% RSLogix 500 project filling_station.RSS, saved by version 8.30.00.16 %
PROJECT "UNTITLED"    % processor: Bul.1763 MicroLogix 1100 Series B %

PROGRAM FILES
  LAD 2   4 rungs
  LAD 3 "IO"  8 rungs
  LAD 4 "STATE"  7 rungs
  LAD 5 "CONTROLS"  4 rungs

DATA FILES
  O0 OUTPUT  4 elements
  I1 INPUT  6 elements
  S2 STATUS  66 elements
  B3 BINARY  3 elements
  T4 TIMER  1 elements
  C5 COUNTER  1 elements
  R6 CONTROL  1 elements
  N7 INTEGER  10 elements
  F8 FLOAT  1 elements

LADDER 2
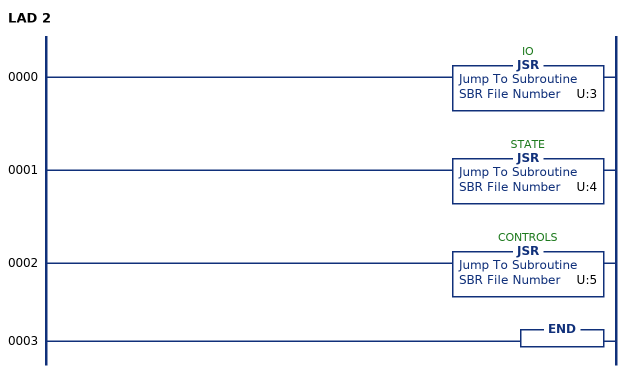
% Rung: 0 %
SOR JSR U:3 EOR
%   U:3  "IO" %
% Rung: 1 %
SOR JSR U:4 EOR
%   U:4  "STATE" %
% Rung: 2 %
SOR JSR U:5 EOR
%   U:5  "CONTROLS" %
% Rung: 3 %
SOR END EOR

LADDER 3 "IO"
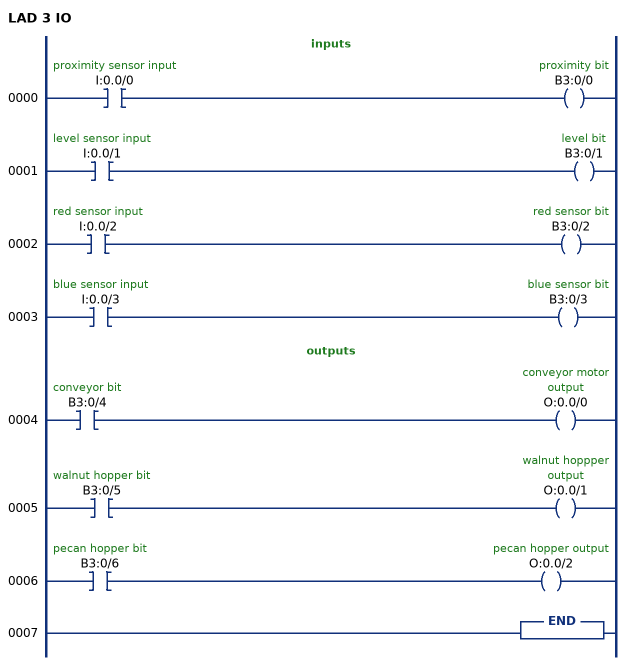
% Rung: 0 %
% TITLE: inputs %
SOR XIC I:0.0/0 OTE B3:0/0 EOR
%   I:0.0/0  "proximity sensor input" %
%   B3:0/0  "proximity bit" %
% Rung: 1 %
SOR XIC I:0.0/1 OTE B3:0/1 EOR
%   I:0.0/1  "level sensor input" %
%   B3:0/1  "level bit" %
% Rung: 2 %
SOR XIC I:0.0/2 OTE B3:0/2 EOR
%   I:0.0/2  "red sensor input" %
%   B3:0/2  "red sensor bit" %
% Rung: 3 %
SOR XIC I:0.0/3 OTE B3:0/3 EOR
%   I:0.0/3  "blue sensor input" %
%   B3:0/3  "blue sensor bit" %
% Rung: 4 %
% TITLE: outputs %
SOR XIC B3:0/4 OTE O:0.0/0 EOR
%   B3:0/4  "conveyor bit" %
%   O:0.0/0  "conveyor motor output" %
% Rung: 5 %
SOR XIC B3:0/5 OTE O:0.0/1 EOR
%   B3:0/5  "walnut hopper bit" %
%   O:0.0/1  "walnut hoppper output" %
% Rung: 6 %
SOR XIC B3:0/6 OTE O:0.0/2 EOR
%   B3:0/6  "pecan hopper bit" %
%   O:0.0/2  "pecan hopper output" %
% Rung: 7 %
SOR END EOR

LADDER 4 "STATE"
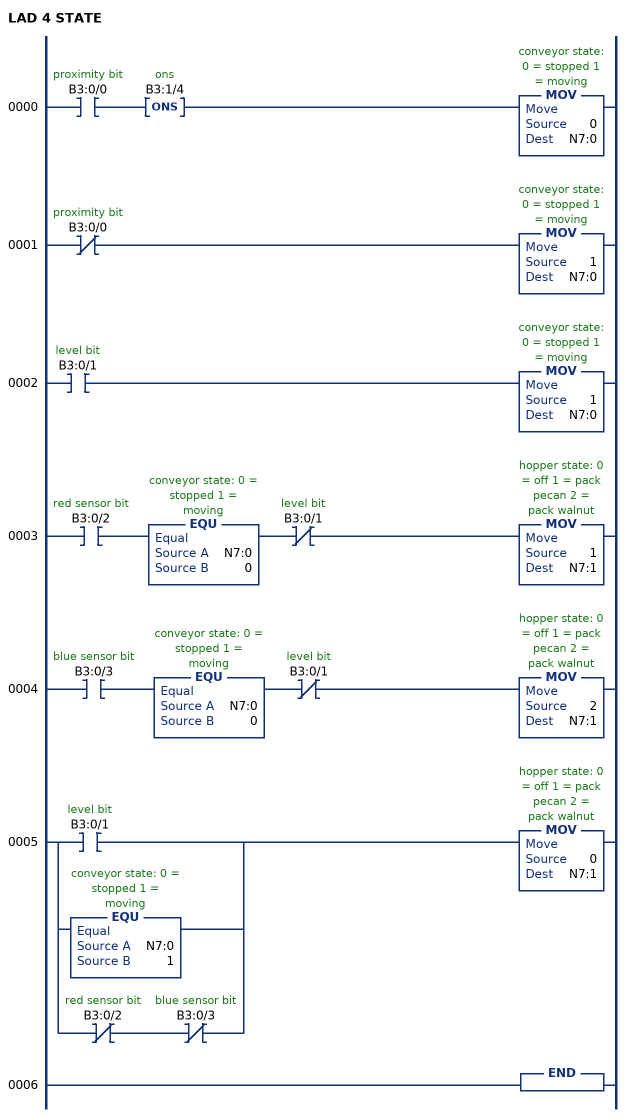
% Rung: 0 %
SOR XIC B3:0/0 ONS B3:1/4 MOV 0 N7:0 EOR
%   B3:0/0  "proximity bit" %
%   B3:1/4  "ons" %
%   N7:0  "conveyor state: 0 = stopped 1 = moving" %
% Rung: 1 %
SOR XIO B3:0/0 MOV 1 N7:0 EOR
%   B3:0/0  "proximity bit" %
%   N7:0  "conveyor state: 0 = stopped 1 = moving" %
% Rung: 2 %
SOR XIC B3:0/1 MOV 1 N7:0 EOR
%   B3:0/1  "level bit" %
%   N7:0  "conveyor state: 0 = stopped 1 = moving" %
% Rung: 3 %
SOR XIC B3:0/2 EQU N7:0 0 XIO B3:0/1 MOV 1 N7:1 EOR
%   B3:0/2  "red sensor bit" %
%   N7:0  "conveyor state: 0 = stopped 1 = moving" %
%   B3:0/1  "level bit" %
%   N7:1  "hopper state: 0 = off 1 = pack pecan 2 = pack walnut" %
% Rung: 4 %
SOR XIC B3:0/3 EQU N7:0 0 XIO B3:0/1 MOV 2 N7:1 EOR
%   B3:0/3  "blue sensor bit" %
%   N7:0  "conveyor state: 0 = stopped 1 = moving" %
%   B3:0/1  "level bit" %
%   N7:1  "hopper state: 0 = off 1 = pack pecan 2 = pack walnut" %
% Rung: 5 %  % edit flag set %
SOR BST XIC B3:0/1 NXB EQU N7:0 1 NXB XIO B3:0/2 XIO B3:0/3 BND MOV 0 N7:1 EOR
%   B3:0/1  "level bit" %
%   N7:0  "conveyor state: 0 = stopped 1 = moving" %
%   B3:0/2  "red sensor bit" %
%   B3:0/3  "blue sensor bit" %
%   N7:1  "hopper state: 0 = off 1 = pack pecan 2 = pack walnut" %
% Rung: 6 %
SOR END EOR

LADDER 5 "CONTROLS"
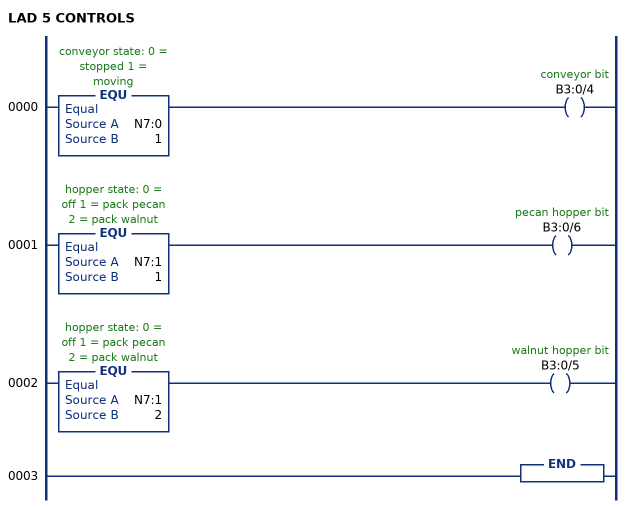
% Rung: 0 %
SOR EQU N7:0 1 OTE B3:0/4 EOR
%   N7:0  "conveyor state: 0 = stopped 1 = moving" %
%   B3:0/4  "conveyor bit" %
% Rung: 1 %
SOR EQU N7:1 1 OTE B3:0/6 EOR
%   N7:1  "hopper state: 0 = off 1 = pack pecan 2 = pack walnut" %
%   B3:0/6  "pecan hopper bit" %
% Rung: 2 %
SOR EQU N7:1 2 OTE B3:0/5 EOR
%   N7:1  "hopper state: 0 = off 1 = pack pecan 2 = pack walnut" %
%   B3:0/5  "walnut hopper bit" %
% Rung: 3 %
SOR END EOR

OTHER DOCUMENTED ADDRESSES
  B3:0/7  "ons"
  B3:0/8  "conveyor trigger"
  B3:0/9  "ons"
  B3:0/10  "conveyor trigger interrupt"
  B3:0/11  "ons"
  B3:0/12  "ons"
  B3:0/13  "ons"
  B3:0/14  "pecan trigger"
  B3:0/15  "walnut trigger"
  B3:1/0  "ons"
  B3:1/1  "packing interrupt"
  B3:1/2  "walnut trigger"
  B3:1/3  "start bit"
  I:0.0/4  "start button"
  N7:0/0  "conveyor state: 0 = stopped 1 = moving"
  N7:0/1  "conveyor state: zero"
  U:6  "CONTROLS"

COMMENTS NOT ATTACHED TO A CURRENT RUNG
  B3:0/14: packing logic
  B3:1/3: inputs

DATA TABLE (non-zero values as saved)
DATA B3
% B3:0 % 0X0201 0X0000 0X0000
